(* PLC project v1.project, CODESYS CODESYS V3.5 SP20 *)
(* stored: creationDateTime 2024-05-17T09:40:45.0541658, modificationDateTime 2024-05-16T13:54:22.2171791 *)

PROGRAM st_1_TON_blink_led
  VAR
    LED : BOOL := FALSE;  (* Variable zur Steuerung der LED *)
    BlinkTimer : TON;  (* Einschaltverzögerung (Timer On) *)
    BlinkInterval : TIME := TIME#1s0ms;  (* Blinkintervall (1 Sekunde) *)
  END_VAR

            // Initialisierung des Timers
BlinkTimer(IN := NOT BlinkTimer.Q, PT := BlinkInterval);

// Logik für das Blinken der LED
IF BlinkTimer.Q THEN
    LED := NOT LED; // LED-Zustand umkehren
END_IF
          
END_PROGRAM

PROGRAM fup_2_XOR_logic
  VAR
    a : BOOL;
    b : BOOL;
    c : BOOL;
    res : BOOL;
  END_VAR

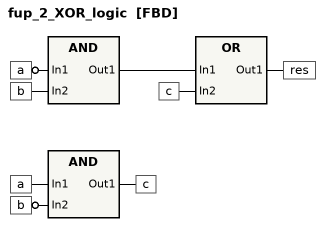
(* FBD diagram, written out as Structured Text *)
res := NOT a AND b OR c;
c := a AND NOT b;
END_PROGRAM

PROGRAM st_3_ARRAY_FOR_IF_bubblesort
  VAR
    arr : ARRAY[1..10] OF INT := [34, 7, 23, 32, 5, 62, 23, 3, 1, 0];  (* Beispiel-Array *)
    n : INT := 10;  (* Größe des Arrays *)
    i : INT;  (* Schleifenvariablen *)
    j : INT;  (* Schleifenvariablen *)
    temp : INT;  (* Temporäre Variable zum Vertauschen *)
    swapped : BOOL;  (* Variable zum Überprüfen, ob Vertauschungen stattgefunden haben *)
  END_VAR

            // Bubble Sort Algorithmus
FOR i := 1 TO n - 1 DO
    swapped := FALSE;
    FOR j := 1 TO n - i DO
        IF arr[j] > arr[j + 1] THEN
            // Vertauschen der Elemente
            temp := arr[j];
            arr[j] := arr[j + 1];
            arr[j + 1] := temp;
            swapped := TRUE;
        END_IF
    END_FOR
    // Wenn keine Vertauschungen stattgefunden haben, ist das Array bereits sortiert
    IF NOT swapped THEN
        EXIT;
    END_IF
END_FOR

// Optional: Ausgabe des sortierten Arrays (abhängig von Ihrer Entwicklungsumgebung)
FOR i := 1 TO n DO
    // Print arr[i]; // Verwenden Sie eine geeignete Methode zur Ausgabe in Ihrer Umgebung
END_FOR
          
END_PROGRAM

PROGRAM fup_1_TON_blink_led
  VAR
    T2 : TON;
    T1 : TON;
    LED : BOOL;
    T2_OUT : BOOL;
  END_VAR

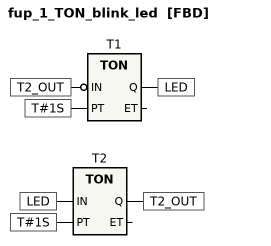
(* FBD diagram, written out as Structured Text *)
T1(IN := NOT T2_OUT, PT := T#1S);
LED := T1.Q;
T2(IN := LED, PT := T#1S);
T2_OUT := T2.Q;
END_PROGRAM

FUNCTION_BLOCK st_1_DIY_BLINKER
  VAR_INPUT
    BlinkInterval : TIME := TIME#1s0ms;  (* Blinkintervall (1 Sekunde) *)
  END_VAR
  VAR_OUTPUT
    Q : BOOL := FALSE;
  END_VAR
  VAR
    BlinkTimer : TON;  (* Einschaltverzögerung (Timer On) *)
  END_VAR

            // Initialisierung des Timers
BlinkTimer(IN := NOT BlinkTimer.Q, PT := BlinkInterval);

// Logik für das Blinken der LED
IF BlinkTimer.Q THEN
    Q := NOT Q; // LED-Zustand umkehren
END_IF
          
END_FUNCTION_BLOCK

PROGRAM fup_1_1_diy_blinker_test
  VAR
    temp : st_1_DIY_BLINKER;
    led_out : BOOL;
  END_VAR

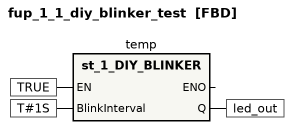
(* FBD diagram, written out as Structured Text *)
temp(EN := TRUE, BlinkInterval := T#1S, Q => led_out);
END_PROGRAM
